// TIA Portal V19 export
DATA_BLOCK "PPrgArchive8"   // DB506
// stored: IsOnlyStoredInLoadMemory true, MemoryReserve 0, Namespace G
   VAR RETAIN
      PRG : Array[701..800] of "PPrg_Data";
   END_VAR
BEGIN
END_DATA_BLOCK
